// TIA Portal V19 export
TYPE "MES_Msg_Receive_Topic4xx_Err"
// stored: Access Published
   STRUCT
      Recive_MSG401 { ExternalAccessible := 'False'; ExternalVisible := 'False'; ExternalWritable := 'False'} : "MES_Err_&_Msg";
      Recive_MSG402 { ExternalAccessible := 'False'; ExternalVisible := 'False'; ExternalWritable := 'False'} : "MES_Err_&_Msg";
      Recive_MSG403 { ExternalAccessible := 'False'; ExternalVisible := 'False'; ExternalWritable := 'False'} : "MES_Err_&_Msg";
      Recive_MSG410 { ExternalAccessible := 'False'; ExternalVisible := 'False'; ExternalWritable := 'False'} : "MES_Err_&_Msg";
      Recive_MSG412 { ExternalAccessible := 'False'; ExternalVisible := 'False'; ExternalWritable := 'False'} : "MES_Err_&_Msg";
      Recive_MSG422 { ExternalAccessible := 'False'; ExternalVisible := 'False'; ExternalWritable := 'False'} : "MES_Err_&_Msg";
      Send_MSG411_Follow_MSG410 { ExternalAccessible := 'False'; ExternalVisible := 'False'; ExternalWritable := 'False'} : "MES_Err_&_Msg";
      Send_MSG413_Follow_MSG412 { ExternalAccessible := 'False'; ExternalVisible := 'False'; ExternalWritable := 'False'} : "MES_Err_&_Msg";
      Send_MSG423_Follow_MSG422 { ExternalAccessible := 'False'; ExternalVisible := 'False'; ExternalWritable := 'False'} : "MES_Err_&_Msg";
   END_STRUCT;
END_TYPE
